// LS Electric XG5000 project: pc로 미니 plc 코일제어
// PLC LSPLC

PROGRAM NewProgram (task: 스캔 프로그램)

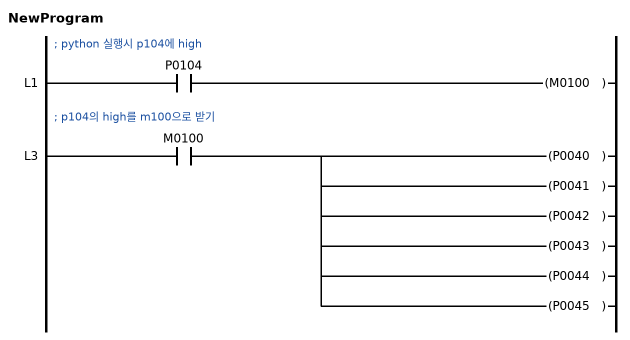
// python 실행시 p104에 high
; L1
LOAD      P0104
OUT       M0100
// p104의 high를 m100으로 받기
; L3
LOAD      M0100
OUT       P0040
OUT       P0041
OUT       P0042
OUT       P0043
OUT       P0044
OUT       P0045